(* PLC project Unnamed, Unknown Unnamed 1 *)
(* stored: creationDateTime 2022-08-16T15:49:17, modificationDateTime 2024-04-03T10:23:07 *)

PROGRAM MQTT_Example
  VAR
    blink_led : BOOL;
    TON0 : TON;
    TOF0 : TOF;
    MQTT_CONNECT0 : MQTT_CONNECT;
    MQTT_SEND0 : MQTT_SEND;
    mqtt_connected : BOOL := 0;
    mqtt_subscribed : BOOL := 0;
    mqtt_sent : BOOL := 0;
    mqtt_received : BOOL := 0;
    msg_received : STRING;
    MQTT_SUBSCRIBE0 : MQTT_SUBSCRIBE;
    MQTT_RECEIVE0 : MQTT_RECEIVE;
  END_VAR
  VAR  (* added by the conversion: wires and edge detectors of the diagram *)
    R_TRIG1 : R_TRIG;
    R_TRIG2 : R_TRIG;
    R_TRIG3 : R_TRIG;
  END_VAR

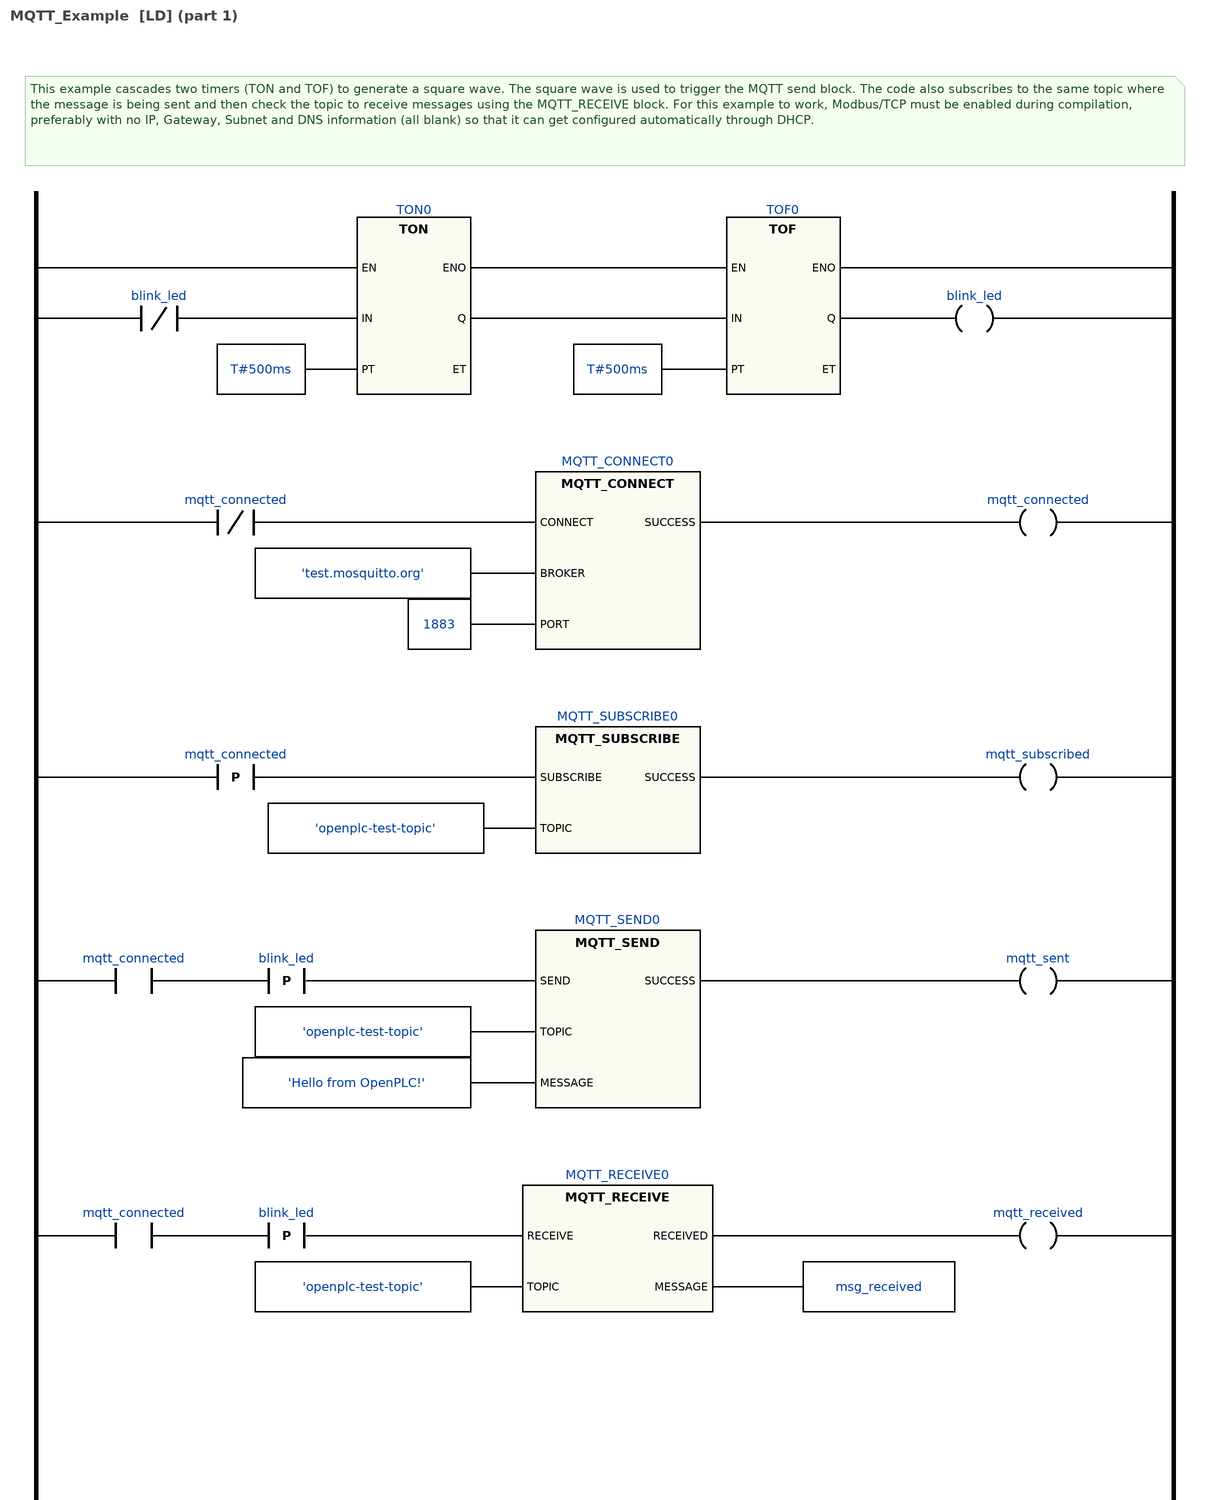
(* LD diagram, written out as Structured Text *)
(* This example cascades two timers (TON and TOF) to generate a square wave. The square wave is used to trigger the MQTT send block. The code also subscribes to the same topic where the message is being sent and then check the topic to receive messages using the MQTT_RECEIVE block. For this example to work, Modbus/TCP must be enabled during compilation, preferably with no IP, Gateway, Subnet and DNS information (all blank) so that it can get configured automatically through DHCP. *)
TON0(IN := NOT blink_led, PT := T#500ms);
TOF0(EN := TON0.ENO, IN := TON0.Q, PT := T#500ms);
blink_led := TOF0.Q;
MQTT_CONNECT0(CONNECT := NOT mqtt_connected, BROKER := 'test.mosquitto.org', PORT := 1883);
mqtt_connected := MQTT_CONNECT0.SUCCESS;
R_TRIG1(CLK := blink_led);
MQTT_SEND0(SEND := mqtt_connected AND R_TRIG1.Q, TOPIC := 'openplc-test-topic', MESSAGE := 'Hello from OpenPLC!');
mqtt_sent := MQTT_SEND0.SUCCESS;
R_TRIG2(CLK := mqtt_connected);
MQTT_SUBSCRIBE0(SUBSCRIBE := R_TRIG2.Q, TOPIC := 'openplc-test-topic');
mqtt_subscribed := MQTT_SUBSCRIBE0.SUCCESS;
R_TRIG3(CLK := blink_led);
MQTT_RECEIVE0(RECEIVE := mqtt_connected AND R_TRIG3.Q, TOPIC := 'openplc-test-topic');
mqtt_received := MQTT_RECEIVE0.RECEIVED;
msg_received := MQTT_RECEIVE0.MESSAGE;
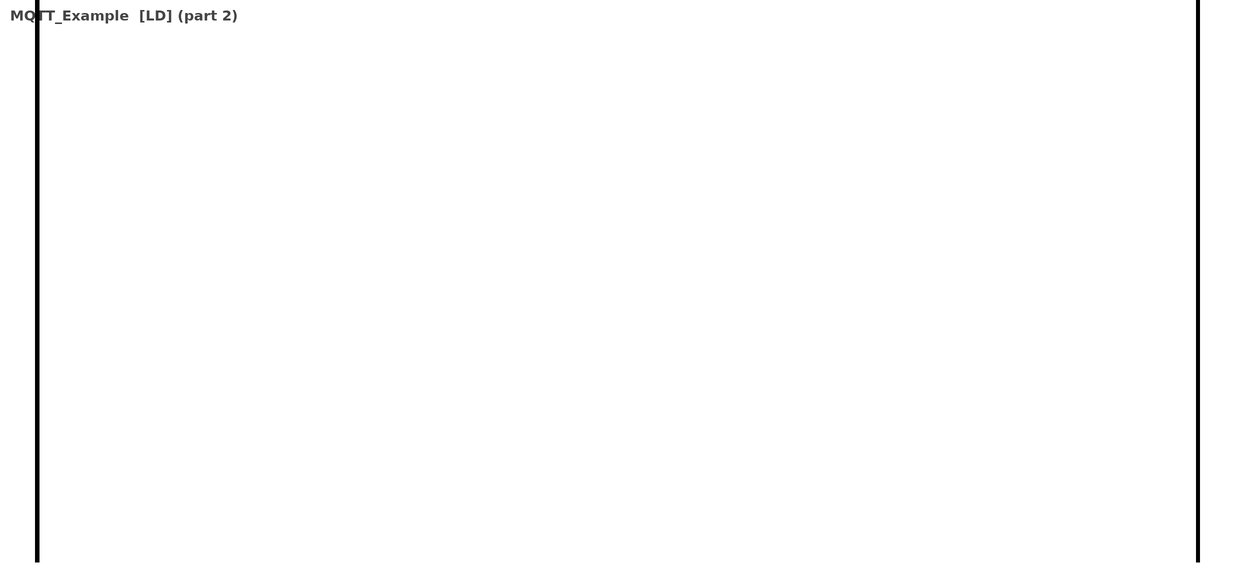
END_PROGRAM

CONFIGURATION Config0
  RESOURCE Res0 ON PLC
    TASK task0(INTERVAL := T#20ms, PRIORITY := 0);
    PROGRAM instance0 WITH task0 : MQTT_Example;
  END_RESOURCE
END_CONFIGURATION
